// TwinCAT 3 PLC project Prog_Eurobot_2020
// ProgramVersion: 3.1.4022.7
// libraries:
//   Tc2_Standard, * (Beckhoff Automation GmbH)
//   Tc2_System, * (Beckhoff Automation GmbH)
//   Tc3_Module, * (Beckhoff Automation GmbH)
// project tree:
//   DUTs/ e_Displacement.TcDUT, e_Type_Action.TcDUT, st_Action.TcDUT
//   FBs/ arrActions.TcPOU, FB_Actions.TcPOU, FB_Beacon.TcPOU, FB_Calcul_Position_V4.TcPOU, FB_ChooseAction.TcPOU, FB_Logger.TcPOU, FB_MoveBezier.TcPOU, FB_MoveLinear.TcPOU, FB_OdometryOpponents.TcPOU, FB_PathFinding.TcPOU
//   GVLs/ IO.TcGVL, Motors.TcGVL
//   / PlcTask.TcTTO, Prg_Match.TcPOU
//   POUs/ Init.TcPOU, MAIN.TcPOU, Mobility.TcPOU
// real-time tasks:
//   TASK PlcTask: cycle T#10ms, priority 20, ADS port 350

CONFIGURATION Prog_Eurobot_2020
    RESOURCE PLC ON TwinCAT3
        TASK PlcTask(INTERVAL := T#10ms, PRIORITY := 20);
        PROGRAM MAIN WITH PlcTask : MAIN;
    END_RESOURCE
END_CONFIGURATION

// ---- DUTs/e_Displacement.TcDUT
{attribute 'qualified_only'}
{attribute 'strict'}
TYPE e_Displacement :
(
	eNoDisplacement := 1<<0, eMoveStraight := 1<<1, eBezierCurve := 1<<2, ePathfinding := 1<<3
);
END_TYPE

// ---- DUTs/e_Type_Action.TcDUT
(*
  \file     	e_Type_Action
  \brief     	enum action types
  \author    	Loïc Nicoud
  \modif		Adrien Jaquiéry		<adrienjaquiery13@gmail.com>	
  \version   	1.0
  \date      	2020-04-24
  \details
*)
TYPE e_Type_Action :
(
	eNull, eDeplacement, eWait, ePushShip, eCheckCompass
);
END_TYPE

// ---- DUTs/st_Action.TcDUT
(*
  \file     	st_Action
  \brief     	action struct
  \author    	Loïc Nicoud
  \modif		Adrien Jaquiéry		<adrienjaquiery13@gmail.com>	
  \version   	1.0
  \date      	2020-04-24
  \details
*)
TYPE st_Action :
STRUCT
	//faire un tableau de cette structure, de [0..?], la case 0 donne l'état initial du robot ( position )
	
	strNomAction : STRING;	//Nom de l'action
	iAction : INT;	//EnumAction (type de l'action à effectuer)
	iPrioriteAction : INT;	//0: ne pas faire, 1 priorité min, plus grand, plus priritaire
	iNbXAction : INT;	//Nombre de fois que l'action peut être faite 0<x<=10 , 10 -> infini	
	iNbActionFaite : INT; //Nombre de fois que l'action à été faite
	
	iTypePrerequis : INT; //0: None, 1: all, 2: min one, 3: min half
	ariPrerequis : ARRAY[1..15] OF INT;	//num tableau action des action prerequises. 0 dans une case -> case ignorée
	
	boActionDone : BOOL;
	boActionAttente : BOOL;	//Si l'action à déja été tentée mais echouée
	
	boDeplacement : BOOL; // True if the action need a displacement
	boPathfinding : bool;
	//Position of the action (if specific position needed)
	lrPosX : LREAL;
	lrPosY : LREAL;
	lrAngle : LREAL;
	
	intPtAction : INT;
	
END_STRUCT
END_TYPE

// ---- GVLs/IO.TcGVL
{attribute 'qualified_only'}
VAR_GLOBAL
	ibStart AT %I*: BOOL;
	ibHome AT %I*: BOOL;
	ibReset AT %I*: BOOL;
	ibAuNc AT %I*: BOOL;
	ibReedStart AT %I*: BOOL;
	
	qbLed1 AT %Q*: BOOL;
	qbLed2 AT %Q*: BOOL;
	qbLed3 AT %Q*: BOOL;
	qbLed4 AT %Q*: BOOL;
END_VAR

// ---- GVLs/Motors.TcGVL
{attribute 'qualified_only'}
VAR_GLOBAL
	motorR: AXIS_REF;
	motorL: AXIS_REF;
	coderR: AXIS_REF;
	coderL: AXIS_REF;
	
	lrPosX: LREAL;
	lrPosY: LREAL;
	lrAngle: LREAL;
	
	
END_VAR

// ---- POUs/MAIN.TcPOU
(*
  \file     	MAIN
  \brief     	main program
  \author    	Adrien Jaquiéry		<adrienjaquiery13@gmail.com>
  \version   	1.0
  \date      	2020-04-24
  \details
*)
PROGRAM MAIN
VAR
	Logger: FB_LOGGER;
	Beacon: FB_Beacon;
	CalculPosition: FB_Calcul_Position_V4;
	
	RtStart: R_TRIG;
	FtStart: F_TRIG;
	FtReset: F_TRIG;
	RtReset: R_TRIG;
	FtHome: F_TRIG;
	RtHome: R_TRIG;
	actions : ARRAY[0..10] OF st_Action;
END_VAR

FtStart(CLK:= IO.ibStart, Q=> );
RtStart(CLK:= IO.ibStart, Q=> );
FtReset(CLK:= IO.ibReset, Q=> );
RtReset(CLK:= IO.ibReset, Q=> );
FtHome(CLK:= IO.ibHome, Q=> );
RtHome(CLK:= IO.ibHome, Q=> );

IF RtReset.Q THEN
	Init();
END_IF

actions := arrActions();


Logger(
	lrPosX:= Motors.lrPosX, 
	lrPosY:= Motors.lrPosY, 
	lrAngle:= Motors.lrAngle, 
	boMovement:= , 
	lrTargetX:= , 
	lrTargetY:= , 
	lrTargetAngle:= , 
	RightMotor:= , 
	LeftMotor:= , 
	RightEncoder:= , 
	LeftEncoder:= , 
	input:= , 
	boMatchEnCours:= IO.ibStart);
	
Beacon(lrDetectionAngle:= , lrMinDistance:= , boFrontDetection:= , boObstacle=> );
(*
CalculPosition(
	lrPosCodeurDroite:= , 
	lrPosCodeurGauche:= , 
	lrEntraxeCodeur:= , 
	boSetPosInitiale:= , 
	lrPosInitialeX:= , 
	lrPosInitialeY:= , 
	lrPosInitialeAngle:= , 
	lrPosActuelleX=> Motors.lrPosX, 
	lrPosActuelleY=> motors.lrPosY, 
	lrPosActuelleAngle=> motors.lrAngle);
	*)

END_PROGRAM

// ---- FBs/FB_Logger.TcPOU
FUNCTION_BLOCK FB_Logger
VAR_INPUT
	lrPosX : LREAL;
	lrPosY : LREAL;
	lrAngle : LREAL;
	
	boMovement : BOOL;			// True if robot is moving
	lrTargetX : LREAL;
	lrTargetY : LREAL;
	lrTargetAngle : LREAL;
	
	eAction : e_Type_Action;			// Current mission type
	
	input : ARRAY[1..10] OF BOOL;	// Inputs for sensors...
	
	RightMotor : AXIS_REF;
	LeftMotor : AXIS_REF;
	RightEncoder : AXIS_REF;
	LeftEncoder : AXIS_REF;
	
	boMatchEnCours : BOOL;
	boReset : bool;
END_VAR
VAR_OUTPUT
END_VAR
VAR
	OpenFile: FB_FileOpen;
	GetTime: NT_GetTime;
	currentTime: TIMESTRUCT;
	path: string;
	TonMatch: TON;
	WriteData: FB_FileWrite;
	logFIle: UINT;
	logText: STRING(250);
	header: STRING;
	boLogData: BOOL;
	WriteHeader: FB_FileWrite;
	CloseFile: FB_FileClose;
	RtStartMatch: R_TRIG;
	boError: BOOL;
	errorId: UDINT;
END_VAR

(*
  \file     	FB_Logger
  \brief     	Log match data in a file
  \author    	Adrien Jaquiéry		<adrienjaquiery13@gmail.com>
  \version   	1.0
  \date      	2020-04-24
  \details
*)
IF boReset = TRUE THEN
	currentTime.wYear := 0;
	boMatchEnCours := FALSE;
	logFIle := 0;
END_IF

RtStartMatch(CLK:= boMatchEnCours, Q=> );
	GetTime(
	NETID:= , 
	START:= boMatchEnCours, 
	TMOUT:= DEFAULT_ADS_TIMEOUT, 
	BUSY=> , 
	ERR=> , 
	ERRID=> , 
	TIMESTR=> currentTime);

	
IF currentTime.wYear <> 0 AND logFIle = 0 AND boMatchEnCours THEN
	path := CONCAT(CONCAT(CONCAT(CONCAT(CONCAT(WORD_TO_STRING(currentTime.wYear),WORD_TO_STRING(currentTime.wMonth)),WORD_TO_STRING(currentTime.wDay)),WORD_TO_STRING(currentTime.wHour)),WORD_TO_STRING(currentTime.wMinute)),WORD_TO_STRING(currentTime.wSecond));

	OpenFile(
		sNetId:= '', 
		sPathName:= CONCAT(path,'.txt'),
		nMode:= FOPEN_MODEWRITE OR FOPEN_MODEPLUS OR FOPEN_MODETEXT, 
		ePath:= PATH_GENERIC, 
		bExecute:= boMatchEnCours, 
		tTimeout:= T#3S, 
		bBusy=> , 
		bError=> boError, 
		nErrId=> errorId, 
		hFile=> logFIle);
END_IF

TonMatch(IN:= boMatchEnCours, PT:= T#100S, Q=> , ET=> );

IF(logFile <> 0 AND boMatchEnCours and not OpenFile.bBusy) THEN
	logText:= CONCAT(CONCAT(CONCAT(CONCAT(CONCAT(CONCAT(TIME_TO_STRING(TonMatch.ET),' posX: '),LREAL_TO_STRING(lrPosX)),' posY: '),LREAL_TO_STRING(lrPosY)),' angle: '),LREAL_TO_STRING(lrAngle));
	logText:= CONCAT(CONCAT(CONCAT(CONCAT(CONCAT(CONCAT(CONCAT(CONCAT(logText,' Mvm: '),BOOL_TO_STRING(boMovement)),' TargetX: '),LREAL_TO_STRING(lrTargetX)),' TargetY: '),LREAL_TO_STRING(lrTargetY)),' TargetAngle: '),LREAL_TO_STRING(lrTargetAngle));
	logText:= CONCAT(CONCAT(logText,' Mission: '),INT_TO_STRING(eAction));
	logText:= CONCAT(CONCAT(CONCAT(CONCAT(CONCAT(CONCAT(CONCAT(CONCAT(CONCAT(CONCAT(CONCAT(CONCAT(CONCAT(CONCAT(CONCAT(CONCAT(CONCAT(CONCAT(CONCAT(CONCAT(logText,' I1: '),BOOL_TO_STRING(input[1])),' I2: '),BOOL_TO_STRING(input[2])),' I3: '),BOOL_TO_STRING(input[3])),' I4: '),BOOL_TO_STRING(input[4])),' I5: '),BOOL_TO_STRING(input[5])),' I6: '),BOOL_TO_STRING(input[6])),' I7: '),BOOL_TO_STRING(input[7])),' I8: '),BOOL_TO_STRING(input[8])),' I9: '),BOOL_TO_STRING(input[9])),' I10: '),BOOL_TO_STRING(input[10]));
	logText:= CONCAT(CONCAT(CONCAT(CONCAT(CONCAT(CONCAT(CONCAT(CONCAT(logText,' rAxErr: '),UDINT_TO_STRING(RightMotor.Status.ErrorID)),' lAxErr: '),UDINT_TO_STRING(leftMotor.Status.ErrorID)),' rIncErr: '),UDINT_TO_STRING(Rightencoder.Status.ErrorID)),' lIncErr: '),UDINT_TO_STRING(Leftencoder.Status.ErrorID));
	logText:= CONCAT(logText,'\n');
	
	WriteData(
	sNetId:= '', 
	hFile:= logFIle, 
	pWriteBuff:= ADR(logText), 
	cbWriteLen:= SIZEOF(logText), 
	bExecute:= NOT boLogData, 
	tTimeout:= , 
	bBusy=> , 
	bError=> boError, 
	nErrId=> errorId, 
	cbWrite=> );
		
END_IF

IF (logFIle <> 0 AND NOT boMatchEnCours) OR CloseFile.bBusy THEN
	CloseFile(
	sNetId:= '', 
	hFile:= logFile, 
	bExecute:= NOT boMatchEnCours AND logFile <> 0, 
	tTimeout:= , 
	bBusy=> , 
	bError=> boError, 
	nErrId=> errorId);	
END_IF

END_FUNCTION_BLOCK

// ---- FBs/FB_Beacon.TcPOU
FUNCTION_BLOCK FB_Beacon
VAR_INPUT
	lrDetectionAngle: LREAL;		// Scaning cone of the beacon. [°](Angle from the front of the robot)
	lrMinDistance: LREAL;		// Minimal distance of detection [mm]
	boFrontDetection: BOOL;		// True = front detection, False = back detection
END_VAR
VAR_OUTPUT
	boObstacle: BOOL;
END_VAR
VAR
	timeBeaconUpdated: TIME := T#500MS;
	IuliBaliseC AT%I* : ULINT;
	IuliBaliseSigPos AT%I* : ULINT;
	IuliBaliseSigNeg AT%I* : ULINT;
	
	uliBaliseOldC : ULINT;
	uliDifference : ULINT;
	lrAngleDetected : LREAL;
	IuliBaliseSigPosOld: ULINT;
	IuliBaliseSigNegOld: ULINT;
	lrAngleDist: LREAL;
	lrDistance : LREAL;
	lrAngleDistRad : lreal;
	TofBaliseAJour: TOF;
	BoBaliseAJour: BOOL;
END_VAR

IF IuliBaliseC <> uliBaliseOldC THEN
	uliDifference := IuliBaliseC - uliBaliseOldC;
	uliBaliseOldC := IuliBaliseC;
END_IF

IF IuliBaliseSigPos <> IuliBaliseSigPosOld THEN
	lrAngleDetected := (((ULINT_TO_LREAL(IuliBaliseSigPos) - ULINT_TO_LREAL(IuliBaliseC)) / ULINT_TO_LREAL(uliDifference))*360.0) + 70.0;
	IF lrAngleDetected > 360.0 THEN
		lrAngleDetected := lrAngleDetected - 360.0;
	ELSIF lrAngleDetected < 0 THEN
		lrAngleDetected := 360.0 + lrAngleDetected;
	END_IF
	IuliBaliseSigPosOld := IuliBaliseSigPos;
END_IF

IF IuliBaliseSigNeg <> IuliBaliseSigNegOld THEN
	lrAngleDist := ((ULINT_TO_LREAL(IuliBaliseSigNeg)- ULINT_TO_LREAL(IuliBaliseSigPos))/ ULINT_TO_LREAL(uliDifference))*360.0;
	lrAngleDistRad := lrAngleDist * PI / 180.0;
	lrDistance := 32 / SIN(lrAngleDistRad / 2.0);
	TofBaliseAJour.IN := TRUE;
	IuliBaliseSigNegOld := IuliBaliseSigNeg;
ELSE
	TofBaliseAJour.IN := FALSE;
END_IF

TofBaliseAJour(IN:= , PT:= timeBeaconUpdated, Q=> BoBaliseAJour, ET=> );
IF BoBaliseAJour = TRUE AND lrDistance <= lrMinDistance AND ((boFrontDetection = TRUE AND (lrdetectionAngle / 2 > lrAngleDetected OR 360 - lrdetectionAngle / 2 < lrAngleDetected)) OR (boFrontDetection = FALSE AND (lrAngleDetected <= 180 AND lrAngleDetected >= 180 - lrdetectionAngle / 2 OR lrAngleDetected > 180 AND lrAngleDetected <= 180 + lrdetectionAngle / 2))) THEN
	boObstacle := TRUE;
ELSE
	boObstacle := FALSE;
END_IF

END_FUNCTION_BLOCK

// ---- FBs/FB_Calcul_Position_V4.TcPOU
FUNCTION_BLOCK FB_Calcul_Position_V4
VAR_INPUT

	lrPosCodeurDroite	: LREAL;
	lrPosCodeurGauche	: LREAL;
	lrEntraxeCodeur		: LREAL;

	boSetPosInitiale	: BOOL;
	lrPosInitialeX		: LREAL;
	lrPosInitialeY		: LREAL;
	lrPosInitialeAngle	: LREAL;	// en [°], le 0° vers Y+, sens horaire

END_VAR
VAR_OUTPUT
	
	lrPosActuelleX		: LREAL;
	lrPosActuelleY		: LREAL;
	lrPosActuelleAngle	: LREAL;

END_VAR
VAR
	
	lrPosCodeurDroiteDernierCycle	: LREAL;
	lrPosCodeurGaucheDernierCycle	: LREAL;
	lrPosActuelleAngleRadian		: LREAL;	

	lrDeltaCodeurDroite		: LREAL;
	lrDeltaCodeurGauche		: LREAL;
	
	lrDeltaDistance		: LREAL;
	lrDeltaAngle		: lreal;
	
END_VAR
VAR CONSTANT
	
	lrValeurPi	: LREAL := 3.1415926535897932384626433832795;

END_VAR

//Gestion set pos initiale

IF boSetPosInitiale THEN
	
	lrPosActuelleX := lrPosInitialeX;
	lrPosActuelleY := lrPosInitialeY;
	lrPosActuelleAngle := lrPosInitialeAngle;
	lrPosActuelleAngleRadian := lrPosInitialeAngle * ( lrValeurPi / 180 );
	
	lrPosCodeurDroiteDernierCycle := lrPosCodeurDroite;
	lrPosCodeurGaucheDernierCycle := lrPosCodeurGauche;

END_IF

//Calcul des deltas codeurs

lrDeltaCodeurDroite := lrPosCodeurDroite - lrPosCodeurDroiteDernierCycle;
lrDeltaCodeurGauche := lrPosCodeurGauche - lrPosCodeurGaucheDernierCycle;

//Calcul distance moyenne et angle

lrDeltaDistance	:= ( lrDeltaCodeurDroite + lrDeltaCodeurGauche ) / 2;
lrDeltaAngle	:= ATAN ( ( lrDeltaCodeurGauche - lrDeltaCodeurDroite ) / lrEntraxeCodeur );

//Calcul pos du robot

lrPosActuelleX := lrPosActuelleX + ( lrDeltaDistance * SIN ( lrPosActuelleAngleRadian ) );
lrPosActuelleY := lrPosActuelleY + ( lrDeltaDistance * COS ( lrPosActuelleAngleRadian ) );

lrPosActuelleAngleRadian := lrPosActuelleAngleRadian + lrDeltaAngle;

IF lrPosActuelleAngleRadian < 0 THEN
	
	lrPosActuelleAngleRadian := lrPosActuelleAngleRadian + ( 2.0 * lrValeurPi );
	
ELSIF lrPosActuelleAngleRadian >= ( 2 * lrValeurPi ) THEN
	
	lrPosActuelleAngleRadian := lrPosActuelleAngleRadian - ( 2.0 * lrValeurPi );

END_IF

lrPosActuelleAngle := lrPosActuelleAngleRadian * ( 180 / lrValeurPi );

lrPosCodeurDroiteDernierCycle := lrPosCodeurDroite;
lrPosCodeurGaucheDernierCycle := lrPosCodeurGauche;

END_FUNCTION_BLOCK

// ---- POUs/Init.TcPOU
PROGRAM Init
VAR
END_VAR

// Write your init sequence here

END_PROGRAM

// ---- FBs/arrActions.TcPOU
FUNCTION arrActions : ARRAY[0..10] OF st_Action;
VAR_INPUT
END_VAR
VAR
END_VAR

//	Set up all actions here

// Action 1
arrActions[1].strNomAction := 'Action 1';		// Name of action
arrActions[1].iAction := eDeplacement;			// Type of action
arrActions[1].iPrioriteAction := 1;				// Priority of action
arrActions[1].iNbXAction := 1;					// Nbr of execution
arrActions[1].iTypePrerequis := 0;				// Type of prerequisite
arrActions[1].ariPrerequis[1] := eNULL;			// Prerequisite actions
arrActions[1].lrPosX := 0;						// Position of the action
arrActions[1].lrPosY := 0;						// If x & y == 0
arrActions[1].lrAngle := 0;						// No deplacement is needed
arrActions[1].intPtAction := 0;					// Nbr of points earned
	
// Action 2	
arrActions[2].strNomAction := 'Action 2';		// Name of action
arrActions[2].iAction := eDeplacement;			// Type of action
arrActions[2].iPrioriteAction := 1;				// Priority of action
arrActions[2].iNbXAction := 1;					// Nbr of execution
arrActions[2].iTypePrerequis := 0;				// Type of prerequisite
arrActions[2].ariPrerequis[1] := eNULL;			// Prerequisite actions
arrActions[2].lrPosX := 0;						// Position of the action
arrActions[2].lrPosY := 0;						// If x & y == 0
arrActions[2].lrAngle := 0;						// No deplacement is needed
arrActions[2].intPtAction := 0;					// Nbr of points earned
// Continue for each action
RETURN;

END_FUNCTION

// ---- FBs/FB_Actions.TcPOU
FUNCTION_BLOCK FB_Actions
VAR_INPUT
END_VAR
VAR_OUTPUT
	arrActions: ARRAY[0..10] OF st_Action;
END_VAR
VAR
END_VAR

//	Set up all actions here

// Action 1
arrActions[1].strNomAction := 'Action 1';		// Name of action
arrActions[1].iAction := eDeplacement;			// Type of action
arrActions[1].iPrioriteAction := 1;				// Priority of action
arrActions[1].iNbXAction := 1;					// Nbr of execution
arrActions[1].iTypePrerequis := 0;				// Type of prerequisite
arrActions[1].ariPrerequis[1] := eNULL;			// Prerequisite actions
arrActions[1].lrPosX := 0;						// Position of the action
arrActions[1].lrPosY := 0;						// If x & y == 0
arrActions[1].lrAngle := 0;						// No deplacement is needed
arrActions[1].intPtAction := 0;					// Nbr of points earned
	
// Action 2	
arrActions[2].strNomAction := 'Action 2';		// Name of action
arrActions[2].iAction := eDeplacement;			// Type of action
arrActions[2].iPrioriteAction := 1;				// Priority of action
arrActions[2].iNbXAction := 1;					// Nbr of execution
arrActions[2].iTypePrerequis := 0;				// Type of prerequisite
arrActions[2].ariPrerequis[1] := eNULL;			// Prerequisite actions
arrActions[2].lrPosX := 0;						// Position of the action
arrActions[2].lrPosY := 0;						// If x & y == 0
arrActions[2].lrAngle := 0;						// No deplacement is needed
arrActions[2].intPtAction := 0;					// Nbr of points earned

// Continue for each action

END_FUNCTION_BLOCK

// ---- FBs/FB_ChooseAction.TcPOU
FUNCTION_BLOCK FB_ChooseAction
VAR_INPUT
END_VAR
VAR_OUTPUT
END_VAR
VAR
END_VAR

END_FUNCTION_BLOCK

// ---- FBs/FB_MoveBezier.TcPOU
FUNCTION_BLOCK FB_MoveBezier
VAR_INPUT
END_VAR
VAR_OUTPUT
END_VAR
VAR
END_VAR

END_FUNCTION_BLOCK

// ---- FBs/FB_MoveLinear.TcPOU
FUNCTION_BLOCK FB_MoveLinear
VAR_INPUT
END_VAR
VAR_OUTPUT
END_VAR
VAR
END_VAR

END_FUNCTION_BLOCK

// ---- FBs/FB_OdometryOpponents.TcPOU
FUNCTION_BLOCK FB_OdometryOpponents
VAR_INPUT
END_VAR
VAR_OUTPUT
END_VAR
VAR
END_VAR

END_FUNCTION_BLOCK

// ---- FBs/FB_PathFinding.TcPOU
FUNCTION_BLOCK FB_PathFinding
VAR_INPUT
END_VAR
VAR_OUTPUT
END_VAR
VAR
END_VAR

END_FUNCTION_BLOCK

// ---- POUs/Mobility.TcPOU
PROGRAM Mobility
VAR
END_VAR

END_PROGRAM

// ---- Prg_Match.TcPOU

PROGRAM Prg_Match
VAR
	
	boChoisirAction: BOOL;
	intChoixAction: INT;
	i: INT;
	intPrioMaxTrouvee: INT;
	boVerifPrerequis: BOOL;
	j: INT;
	intVerifAction: USINT;
	intNbActionVerifTot: INT;
	intNbActionVerifDone: INT;
	TON_1 : TON;
	boVerifPucAttente: BOOL;
	intNbPucsPris: INT;
	intNbPucDansRobot: INT;
	boGoldPris: BOOL;
	R_TRIG_StartMove: R_TRIG;
	R_TRIG_Depl: R_TRIG;
	R_TRIG_Algo: R_TRIG;
	TON_2: TON;
	R_TRIG_Move: R_TRIG;
	ADSREAD_1: ADSREAD;
	boResetExp : BOOL := TRUE;
	ADSWRITE_1: ADSWRITE;
	TON_Blink1: TON;
	TON_Blink2: TON;
	ADSWRITE_2: ADSWRITE;
	boDesactiverExp: BOOL := FALSE;;
	boEtatReset: BOOL;
	ADSREAD_2: ADSREAD;
	TON_reset: TON;
	R_TRIG_Etape: R_TRIG;
	NbPucsBalance: INT;
	bRenewDeplEv: BOOL;
	boLireEtatExp: BOOL;
	ADSREAD_3: ADSREAD;
	R_TRIG_Agold: R_TRIG;
	R_TRIG_APousser: R_TRIG;
	R_TRIG_Aok : R_TRIG;
	test: BOOL;
	attentefront: BOOL;
END_VAR

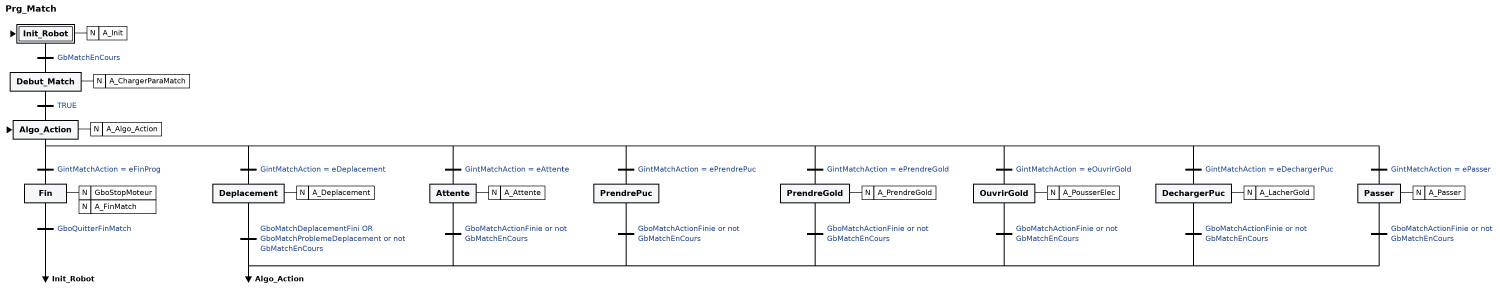
INITIAL_STEP Init_Robot:
    A_Init(N);
END_STEP
TRANSITION FROM Init_Robot TO Debut_Match
    := GbMatchEnCours;
END_TRANSITION
STEP Debut_Match:
    A_ChargerParaMatch(N);
END_STEP
TRANSITION FROM Debut_Match TO Algo_Action
    := TRUE;
END_TRANSITION
STEP Algo_Action:
    A_Algo_Action(N);
END_STEP
TRANSITION FROM Algo_Action TO Fin
    := GintMatchAction = eFinProg;
END_TRANSITION
STEP Fin:
    GboStopMoteur(N);
    A_FinMatch(N);
END_STEP
TRANSITION FROM Fin TO Init_Robot
    := GboQuitterFinMatch;
END_TRANSITION
TRANSITION FROM Algo_Action TO Deplacement
    := GintMatchAction = eDeplacement;
END_TRANSITION
STEP Deplacement:
    A_Deplacement(N);
END_STEP
TRANSITION FROM Deplacement TO Algo_Action
    := GboMatchDeplacementFini OR GboMatchProblemeDeplacement or not GbMatchEnCours;
END_TRANSITION
TRANSITION FROM Algo_Action TO Attente
    := GintMatchAction = eAttente;
END_TRANSITION
STEP Attente:
    A_Attente(N);
END_STEP
TRANSITION FROM Attente TO Algo_Action
    := GboMatchActionFinie or not GbMatchEnCours;
END_TRANSITION
TRANSITION FROM Algo_Action TO PrendrePuc
    := GintMatchAction = ePrendrePuc;
END_TRANSITION
STEP PrendrePuc:
END_STEP
TRANSITION FROM PrendrePuc TO Algo_Action
    := GboMatchActionFinie or not GbMatchEnCours;
END_TRANSITION
TRANSITION FROM Algo_Action TO PrendreGold
    := GintMatchAction = ePrendreGold;
END_TRANSITION
STEP PrendreGold:
    A_PrendreGold(N);
END_STEP
TRANSITION FROM PrendreGold TO Algo_Action
    := GboMatchActionFinie or not GbMatchEnCours;
END_TRANSITION
TRANSITION FROM Algo_Action TO OuvrirGold
    := GintMatchAction = eOuvrirGold;
END_TRANSITION
STEP OuvrirGold:
    A_PousserElec(N);
END_STEP
TRANSITION FROM OuvrirGold TO Algo_Action
    := GboMatchActionFinie or not GbMatchEnCours;
END_TRANSITION
TRANSITION FROM Algo_Action TO DechargerPuc
    := GintMatchAction = eDechargerPuc;
END_TRANSITION
STEP DechargerPuc:
    A_LacherGold(N);
END_STEP
TRANSITION FROM DechargerPuc TO Algo_Action
    := GboMatchActionFinie or not GbMatchEnCours;
END_TRANSITION
TRANSITION FROM Algo_Action TO Passer
    := GintMatchAction = ePasser;
END_TRANSITION
STEP Passer:
    A_Passer(N);
END_STEP
TRANSITION FROM Passer TO Algo_Action
    := GboMatchActionFinie or not GbMatchEnCours;
END_TRANSITION

ACTION A_Algo_Action:
R_TRIG_Algo(Clk := Algo_Action.x);

boSetPosInitiale := FALSE;

IF R_TRIG_Algo.Q THEN
	//Algorithme Action
	IF GboMatchDebutMatch THEN
		GboMatchDebutMatch := FALSE;
		boChoisirAction := TRUE;
	ELSIF GboMatchDeplacementFini THEN
		GboMatchDeplacementFini := FALSE;
		GintMatchAction := GarstMatchParaMatch[intChoixAction].uiAction;
	ELSIF GboMatchProblemeDeplacement THEN
		GboMatchProblemeDeplacement := FALSE;
		GarstMatchParaMatch[intChoixAction].boActionAttente := TRUE;
		boChoisirAction := TRUE;
	ELSIF GboMatchActionFinie THEN
	
		GboMatchActionFinie := FALSE;
		
		IF GintMatchAction <> eAttente THEN
			GarstMatchParaMatch[intChoixAction].uiNbActionFaite := GarstMatchParaMatch[intChoixAction].uiNbActionFaite + 1;	//incrmeneter le nb de fois que l'action a ete faite
			
			GNombrePointsMatch := GNombrePointsMatch + GarstMatchParaMatch[intChoixAction].intPtAction;	//increment des point de l'action qui vient d'etre aite
		
			IF GarstMatchParaMatch[intChoixAction].uiNbActionFaite >= GarstMatchParaMatch[intChoixAction].uiNbXAction AND GarstMatchParaMatch[intChoixAction].uiNbXAction <> 10 THEN
				GarstMatchParaMatch[intChoixAction].boActionDone := TRUE;
			END_IF
		END_IF
		boChoisirAction := TRUE;
		
		//Remmetre a false les action en attente
		FOR i := 1 TO GintMatchNoActionMax DO
			GarstMatchParaMatch[i].boActionAttente := FALSE;
		END_FOR
		
		
		//--------------------------------------------
		IF intChoixAction = 2 THEN
			boGoldPris := TRUE;
		END_IF
		
		IF (( 2 <= intChoixAction ) AND ( intChoixAction <= 14 )) and (GintMatchAction <> eAttente) THEN //si un pucs a ete pris, incrementer les nb de pucs dans le robot
			intNbPucDansRobot := intNbPucDansRobot + 1;
		ELSIF intChoixAction = 15 THEN	//si les pucs ont ete posé, remettre a 0 le nb de pucs dans le robot
			intNbPucDansRobot := 0;
			boGoldPris := FALSE;
		END_IF
	END_IF
	
	//-------------------------------------------------------------------------------------
	//Inserer ici moulinette algorithmique pouzr certianes actions non normales
		//Les action 28 a 30 permette de gerer quand on peut prendre / poser des pucs normaux
	//-----------------------------------------------------------------------------------------
	
	

	//------------------------------------------------------------------------------------------------
	//------------------------------------------------------------------------------------------------
	//Choix action
	
	intPrioMaxTrouvee := -1;
	
	IF boChoisirAction THEN
		boChoisirAction := FALSE;
		
		//trouver l'action la plus prioritaire possible
		FOR i := 1 TO GintMatchNoActionMax DO
			IF GarstMatchParaMatch[i].uiPrioriteAction > intPrioMaxTrouvee THEN
				//Verifier quelle peut etre faite
				IF NOT ( GarstMatchParaMatch[i].boActionDone ) AND NOT ( GarstMatchParaMatch[i].boActionAttente ) THEN
					CASE GarstMatchParaMatch[i].usiTypePrerequis OF
						0:	//Pas de prerequis
								//-> nouveau max 
							intChoixAction := i;
							intPrioMaxTrouvee := GarstMatchParaMatch[i].uiPrioriteAction;
							
						1:	//Verifier tous les prerequis
							boVerifPrerequis := TRUE;
							
							FOR j := 1 TO 15 DO
								intVerifAction := GarstMatchParaMatch[i].arusiPrerequis[j];
								IF intVerifAction <> 0 THEN
									IF NOT GarstMatchParaMatch[intVerifAction].boActionDone THEN
										boVerifPrerequis := FALSE;
									END_IF
								END_IF
							END_FOR
							
							IF boVerifPrerequis THEN
								intChoixAction := i;
								intPrioMaxTrouvee := GarstMatchParaMatch[i].uiPrioriteAction;
							END_IF
							
						2:	//Verifier si au moin un prerequis et fait
							intNbActionVerifTot := 0;
							intNbActionVerifDone := 0;
							
							FOR j := 1 TO 15 DO
								intVerifAction := GarstMatchParaMatch[i].arusiPrerequis[j];
								IF intVerifAction <> 0 THEN
										intNbActionVerifTot := intNbActionVerifTot + 1;
										IF GarstMatchParaMatch[intVerifAction].boActionDone THEN
											intNbActionVerifDone := intNbActionVerifDone + 1;
										END_IF
								END_IF							
							END_FOR
							
							IF intNbActionVerifDone >= ( intNbActionVerifTot / 2 ) THEN
								intChoixAction := i;
								intPrioMaxTrouvee := GarstMatchParaMatch[i].uiPrioriteAction;
							END_IF
							
						3:	//Verifier si tout les prerequis sont fait
							intNbActionVerifTot := 0;
							intNbActionVerifDone := 0;
							
							FOR j := 1 TO 15 DO
								intVerifAction := GarstMatchParaMatch[i].arusiPrerequis[j];
								IF intVerifAction <> 0 THEN
									intNbActionVerifTot := intNbActionVerifTot + 1;
									IF GarstMatchParaMatch[intVerifAction].boActionDone THEN
										intNbActionVerifDone := intNbActionVerifDone + 1;
									END_IF
								END_IF							
							END_FOR
							
							IF intNbActionVerifDone = intNbActionVerifTot THEN
								intChoixAction := i;
								intPrioMaxTrouvee := GarstMatchParaMatch[i].uiPrioriteAction;
							END_IF
					END_CASE
				END_IF
			END_IF
		END_FOR
		
		IF intPrioMaxTrouvee <> -1 THEN
			//action trouvée aller a la position
			GintMatchActionObjectif := intChoixAction;
			GintMatchAction := eDeplacement;
		ELSE
			//pas d'actiopn trouvée, attendre 3s
			GtimeMatchDelayAttendre := T#3S;
			GintMatchAction := eAttente;
		END_IF
	END_IF

	//Cas plus en match
	IF NOT GbMatchEnCours THEN
		GintMatchAction := eFinProg;
	END_IF
END_IF
END_ACTION

ACTION A_Attente:
TON_1(IN:= Attente.x, PT:= GtimeMatchDelayAttendre);

IF TON_1.Q THEN
	GboMatchActionFinie := true;
END_IF
END_ACTION

ACTION A_ChargerParaMatch:
IF Debut_Match.x THEN
	Fn_ViderParaMatch();

	IF GboMatchCouleur THEN
		//violet
		Fn_ChargerParaViolet();
	ELSE
		//jaune
		Fn_ChargerParaJaune();	
	END_IF
	
	GNombrePointsMatch := 5;	//5pt pose experience
	intChoixAction := 0;
	intNbPucDansRobot := 0;
	GboMatchDebutMatch := TRUE;
	boResetCommandeMoteur := FALSE;
	NbPucsBalance := 0;
	boSetPosInitiale := TRUE;
	etat_trajectoire := 1;
	StartDepl := FALSE;
	GarlrObstacles[1,2] := 0;
	GarlrObstacles[1,3] := 0;
	GboPrendreGold := FALSE;
	GboPousserElec := FALSE;
END_IF
END_ACTION

ACTION A_Deplacement:
R_TRIG_Depl(CLK:= Deplacement.x);
R_TRIG_Move(CLK := GboMoveDone);

IF  R_TRIG_Depl.Q THEN
	boReculerDepl := FALSE;
END_IF

IF R_TRIG_Depl.Q OR bRenewDeplEv THEN
	MAIN_1.pt_arrivee := GintMatchActionObjectif;
	etat_trajectoire := 2;
	bRenewDeplEv := FALSE;
	boResetCommandeMoteur := FALSE;
END_IF

R_TRIG_StartMove(CLK :=  etat_trajectoire = 10);

IF R_TRIG_StartMove.Q THEN
	//Deplacement calcul ok
	//PRG_CommandeMoteur.start_move := TRUE;	
	StartDepl := TRUE;
ELSIF etat_trajectoire = 6 THEN
	//Calcul pas ok
	GboMatchProblemeDeplacement := TRUE;
ELSIF etat_trajectoire = 7 THEN
	etat_trajectoire := 2;
ELSIF R_TRIG_Move.Q THEN
	StartDepl := FALSE;
	GboMatchDeplacementFini := TRUE;
ELSIF GbObstacleDerriere AND boSensLigneDroite AND StartDepl AND boEnLigneDroite THEN
	boEnLigneDroite := FALSE;
	boStopMotor := TRUE;
	StartDepl := FALSE;
	GarlrObstacles[1,2] := GlrPosX - 550 * COS(GlrAngle);
	GarlrObstacles[1,3] := GlrPosY - 550 * SIN(GlrAngle);
ELSIF GbObstacleDevant AND NOT boSensLigneDroite AND StartDepl AND boEnLigneDroite THEN
	boEnLigneDroite := FALSE;
	boStopMotor := TRUE;
	StartDepl := FALSE;
	GarlrObstacles[1,2] := GlrPosX + 550 * COS(GlrAngle);
	GarlrObstacles[1,3] := GlrPosY + 550 * SIN(GlrAngle);
ELSIF boStopDoneGc AND boStopDoneDr THEN
	//stop fini, refaire deplacment, reculer de 100
	boReculerDepl := TRUE;
	boStopMotor := FALSE;
	boResetCommandeMoteur := TRUE;
	bRenewDeplEv := TRUE;
END_IF
END_ACTION

ACTION A_FinMatch:
TON_2(IN:= Fin.x , PT:= T#2S);

GboMatchActionFinie := FALSE;
GboMatchDeplacementFini := FALSE;

QboEnableVentDroite := FALSE;
QboEnableVentGauche := FALSE;

GboPrendreGold := FALSE;
GboPousserElec := FALSE;

boStopMotor := TRUE;

IF TON_2.Q THEN
	boPowerMotor := FALSE;
END_IF

GstrMatchNomActionEnCour := 'Fin du match';
END_ACTION

ACTION A_Init:
R_TRIG_Etape(Clk := Init_Robot.x);

IF R_TRIG_Etape.Q THEN
	boResetExp := TRUE;
END_IF

GboQuitterFinMatch := FALSE;

IF GboMatchAuReleve THEN
	boStopMotor := FALSE;
	boPowerMotor := TRUE;
	boResetCommandeMoteur := TRUE;
ELSE
	boPowerMotor := FALSE;
END_IF

//Reset de l'experience
TON_Blink1(IN:= Init_robot.x AND NOT TON_Blink2.Q, PT:= T#1.5S);
TON_Blink2(IN:= TON_Blink1.Q, PT:= T#1.5S);

ADSREAD_2(
	NETID:= '192.168.0.151.1.1', 
	PORT:= 801, 
	IDXGRP:= 16#4020, 
	IDXOFFS:= 102, 
	LEN:= SIZEOF(boEtatReset), 
	DESTADDR:= ADR(boEtatReset), 
	READ:= TON_Blink1.Q, 
	TMOUT:= T#2S, 
	BUSY=> , 
	ERR=> , 
	ERRID=> );

ADSWRITE_1(
	NETID:= '192.168.0.151.1.1', 
	PORT:= 801, 
	IDXGRP:= 16#4020, 
	IDXOFFS:= 102, 
	LEN:= SIZEOF(boResetExp), 
	SRCADDR:= ADR(boResetExp), 
	WRITE:= TON_Blink1.Q, 
	TMOUT:= T#2S, 
	BUSY=> , 
	ERR=> , 
	ERRID=> );

ADSREAD_3(
	NETID:= '192.168.0.151.1.1', 
	PORT:= 801, 
	IDXGRP:= 16#4020, 
	IDXOFFS:= 200, 
	LEN:= SIZEOF(boLireEtatExp), 
	DESTADDR:= ADR(boLireEtatExp), 
	READ:= TON_Blink1.Q, 
	TMOUT:= T#2S, 
	BUSY=> , 
	ERR=> , 
	ERRID=> );
		
TON_reset(IN:= boEtatReset, PT:= T#4S);
IF TON_reset.Q THEN
	boResetExp := FALSE;
END_IF

IF boLireEtatExp THEN
	
	ADSWRITE_2(
		NETID:= '192.168.0.151.1.1', 
		PORT:= 801, 
		IDXGRP:= 16#4020, 
		IDXOFFS:= 100, 
		LEN:= SIZEOF(boDesactiverExp), 
		SRCADDR:= ADR(boDesactiverExp), 
		WRITE:= TON_Blink1.Q, 
		TMOUT:= T#2S, 
		BUSY=> , 
		ERR=> , 
		ERRID=> );
	
	ADSREAD_1(
		NETID:= '192.168.0.151.1.1', 
		PORT:= 801, 
		IDXGRP:= 16#4020, 
		IDXOFFS:= 200, 
		LEN:= SIZEOF(Prog_Activer_Experience.boLireEtatExp), 
		DESTADDR:= ADR(Prog_Activer_Experience.boLireEtatExp), 
		READ:= TON_Blink1.Q, 
		TMOUT:= T#2S, 
		BUSY=> , 
		ERR=> , 
		ERRID=> );
		
END_IF
END_ACTION

ACTION A_LacherGold:
QboEnableVentDroite := FALSE;
QboEnableVentGauche := FALSE;

GboMatchActionFinie := TRUE;
END_ACTION

ACTION A_Passer:
GboMatchActionFinie := TRUE;
END_ACTION

ACTION A_PousserElec:
R_TRIG_APousser( Clk := OuvrirGold.x );

IF R_TRIG_APousser.Q THEN
	GboPousserElec := TRUE;
	IF GboActionok THEN
		attentefront := TRUE;
	ELSE
		attentefront := FALSE;
	END_IF
END_IF

IF NOT GboActionok THEN
	attentefront := FALSE;
END_IF

IF (NOT attentefront) AND GboActionok THEN
	GboPousserElec := FALSE;
	GboMatchActionFinie := TRUE;
END_IF
END_ACTION

ACTION A_PrendreGold:
R_TRIG_Agold( Clk := PrendreGold.x );

IF R_TRIG_Agold.Q THEN
	GboPrendreGold := TRUE;
		IF GboActionok THEN
		attentefront := TRUE;
	ELSE
		attentefront := FALSE;
	END_IF
END_IF

IF NOT GboActionok THEN
	attentefront := FALSE;
END_IF

IF (NOT attentefront) AND GboActionok THEN
	GboPrendreGold := FALSE;
	GboMatchActionFinie := TRUE;
END_IF
END_ACTION

END_PROGRAM
